Staubli VAL3: IoWriteRequestMsg.pjx

--- IoWriteRequestMsg.pjx ---
Parameters version=s7.7.2 stackSize=5000 millimeterUnit=true
Program file=start.pgx
Program file=stop.pgx
Data file=IoWriteRequestMsg.dtx
Type name=IoWriteRequest path=Disk://ros_libs/IoWriteRequest/IoWriteRequest.pjx
Type name=Prefix path=Disk://ros_libs/Prefix/Prefix.pjx
Type name=Header path=Disk://ros_libs/Header/Header.pjx
Type name=Body path=Disk://ros_libs/Body/Body.pjx

--- IoWriteRequestMsg.dtx ---
public Body body
  [0]
    num nData[28]
public Header header
  [0]
    num nMsgType
    num nCommType
    num nReplyCode
    num nData[9]
public Prefix prefix
  [0]
    num nLength
    num nData[4]
public IoWriteRequest ioWriteRequest
  [0]
    num nCount
    num nType
    num nIndex
    num nValue

--- start.pgx ---
program start()
begin
  // Copyright (c) 2016, Ocado Technology - Robotics Research Team
  // Copyright (c) 2019, isys vision
  //
  // Licensed under the Apache License, Version 2.0 (the "License");
  // you may not use this file except in compliance with the License.
  // You may obtain a copy of the License at
  //
  //     http://www.apache.org/licenses/LICENSE-2.0
  //
  // Unless required by applicable law or agreed to in writing, software
  // distributed under the License is distributed on an "AS IS" BASIS,
  // WITHOUT WARRANTIES OR CONDITIONS OF ANY KIND, either express or implied.
  // See the License for the specific language governing permissions and
  // limitations under the License.



end

--- stop.pgx ---
program stop()
begin
  // Copyright (c) 2016, Ocado Technology - Robotics Research Team
  // Copyright (c) 2016, Ocado Technology - Robotics Research Team
  //
  // Licensed under the Apache License, Version 2.0 (the "License");
  // you may not use this file except in compliance with the License.
  // You may obtain a copy of the License at
  //
  //     http://www.apache.org/licenses/LICENSE-2.0
  //
  // Unless required by applicable law or agreed to in writing, software
  // distributed under the License is distributed on an "AS IS" BASIS,
  // WITHOUT WARRANTIES OR CONDITIONS OF ANY KIND, either express or implied.
  // See the License for the specific language governing permissions and
  // limitations under the License.



end
